// base first (§3.14.2); then children, one-shot init, mode transition, stall watch
METHOD PROTECTED OnCyclic : DINT
VAR
    publishIdx : INT;
    modeIdx    : E_Mode;
    styleIdx   : E_RunStyle;
    previousMode : E_Mode;
    modeExitResult : DINT;
END_VAR
OnCyclic := SUPER^.OnCyclic();
_M_TickChildren();
_M_OeeUpdate();                                       // §8.5.1 time accounting + sampling
AlarmLog.Cyclic();                                    // §8.10 shelf auto-expiry
_M_HandleHmiRequest();                                // §3.10 request mailbox
Access.Cyclic();
// §9.8 data-driven Control On/Off request endpoint. Off wins if both arrive;
// the domain/power-group implementation still validates safety, health and rearm.
ControlOnRequest := FALSE;
ControlOffRequest := FALSE;
IF ReqControlOff THEN
    ReqControlOff := FALSE;
    ReqControlOn := FALSE;
    IF Access.PermitsLogged(Gate := E_GatedAction.POWER_CONTROL) THEN
        ControlOffRequest := TRUE;
    END_IF
ELSIF ReqControlOn THEN
    ReqControlOn := FALSE;
    IF Access.PermitsLogged(Gate := E_GatedAction.POWER_CONTROL) THEN
        ControlOnRequest := TRUE;
    END_IF
END_IF
// §3.14.4 — pending mode change; §3.4.1 style decides graceful vs immediate
IF _modePend THEN
    IF _exec = E_ExecState.BUSY THEN
        IF ModePolicy[TO_INT(_mode)].Style = E_ModeSwitchStyle.GRACEFUL THEN
            _stopReq := TRUE;                             // finish the cycle at its stop point
        ELSE
            modeExitResult := OnModeExit(FirstCall := _modeExitFirst,
                RequestedMode := _modeReq);
            _modeExitFirst := FALSE;
            IF modeExitResult = 0 THEN
                OnAbort();                                // IMMEDIATE: cancel now (override may defer)
            END_IF
        END_IF
    ELSE
        IF _exec <> E_ExecState.READY THEN
            Execute := FALSE;                             // release the run command (§6.1 reset)
        ELSE
            previousMode := _mode;
            _mode := _modeReq;
            _modePend := FALSE;
            _modeExitFirst := FALSE;
            _M_CascadeMode(_mode);                        // §3.7 cascade [TC3]
            OnModeChanged(NewMode := _mode, OldMode := previousMode);
        END_IF
    END_IF
END_IF
// §8.3(c) — automatic fault capture: ERROR entry raises, ERROR exit marks gone
IF (_exec = E_ExecState.ERROR) AND (_faultEvt = 0) THEN
    _faultEvt := AlarmLog.RaiseDiag(D := _diag, ResetClass := E_ResetClass.MANUAL_RESET);
    _M_PartAborted();                  // §3.16.3: a faulted part leaves without a valid result
ELSIF (_exec <> E_ExecState.ERROR) AND (_faultEvt > 0) THEN
    AlarmLog.Gone(Slot := _faultEvt);                            // -> WAIT_RESET (blocking)
    _faultEvt := 0;
END_IF
// §6.9 — instant rollup on awaited Error; stall as PENDING otherwise
IF _exec = E_ExecState.BUSY THEN
    IF (_awaits <> 0) AND_THEN _awaits.FaultActive THEN
        _M_FaultDiag(_awaits.GetFaultSummary());
    ELSE
        _tStall(IN := TRUE, PT := SEL(CurrentStep.ExpectedTime > T#0S, StallTime, CurrentStep.ExpectedTime));
        IF _tStall.Q THEN
            _M_StallWalk();
        END_IF
    END_IF
ELSE
    _tStall(IN := FALSE);
END_IF
// §6.9(a) — every new fault joins the shift-change ring, no historian needed
_fTrig(CLK := (_exec = E_ExecState.ERROR));
IF _fTrig.Q THEN
    _M_PushHistory(_diag);
END_IF
// §8.11.4(d) — creeping WORK time is a MAINTENANCE event (Low), not downtime:
// the profiler pulses once per excursion past the configured baseline band.
IF Profiler.DegradedTrig THEN
    _M_RaiseMaintenance(Reason := E_Reason.CYCLE_TIME_DEGRADED,
        Text := 'std.maintenance.cycleTimeDegraded');
END_IF
ModeActivePublished := _mode;
RunningPublished := (_exec = E_ExecState.BUSY);
StopPendingPublished := _stopReq AND (_exec = E_ExecState.BUSY);
FOR publishIdx := 0 TO PL_Fraktal.MODE_COUNT - 1 DO
    modeIdx := publishIdx;
    SupportedModesPublished[publishIdx] := _M_Supports(Mode := modeIdx);
END_FOR
FOR publishIdx := 0 TO 2 DO
    styleIdx := publishIdx;
    SupportedRunStylesPublished[publishIdx] := _M_SupportsRunStyle(Style := styleIdx);
END_FOR
END_METHOD

// §3.14 hook — one-shot after first operational scan
METHOD PROTECTED OnInit : DINT
OnInit := SUPER^.OnInit();
Access.Setup(Provider := 0, pAlarmLog := ADR(AlarmLog)); // preserves an injected provider
_M_InitModePolicy();
// §3.10.2 — seed the manifest revision from boot time so every PLC restart or
// re-activation yields a NEW value (a plain counter would repeat after reboot
// and an HMI could keep a stale manifest undetected). Config writes increment.
ConfigRev := DT_TO_UDINT(F_Now());
END_METHOD

// §3.14 hook — after the new mode is committed
METHOD PROTECTED OnModeChanged : DINT
VAR_INPUT
    NewMode : E_Mode;
    OldMode : E_Mode;
END_VAR
OnModeChanged := 0;
END_METHOD

// §3.14.4 — called every scan while a mode request is pending and the Unit is BUSY.
// Return 0 = consent to immediate cancel (default); >0 = still stopping gracefully.
METHOD PROTECTED OnModeExit : DINT
VAR_INPUT
    FirstCall : BOOL;
    RequestedMode : E_Mode;
END_VAR
OnModeExit := 0;
END_METHOD

// §8.3(b) — deliberate operator reset of blocking events (release-gated per §7.6/§14).
// Closes WAIT_RESET events; an event whose condition persists stays ACTIVE.
METHOD OperatorReset : BOOL
IF NOT Access.PermitsLogged(Gate := E_GatedAction.ALARM_RESET) THEN
    OperatorReset := FALSE;            // §7.7
    RETURN;
END_IF
OperatorReset := AlarmLog.OperatorReset();
END_METHOD

// §3.8 optional HMI/MES selection catalog. Recipe providers remain pluggable;
// the application registers only the model identities it deliberately exposes.
METHOD RegisterAvailableModel : BOOL
VAR_INPUT
    Id : ST_ModelId;
END_VAR
VAR
    i : INT;
END_VAR
RegisterAvailableModel := FALSE;
IF (Id.ModelCode = '') OR (AvailableModelCount >= PL_Fraktal.MAX_RECIPES) THEN
    RETURN;
END_IF
FOR i := 1 TO AvailableModelCount DO
    IF AvailableModels[i].ModelCode = Id.ModelCode THEN
        RETURN;
    END_IF
END_FOR
AvailableModelCount := AvailableModelCount + 1;
AvailableModels[AvailableModelCount] := Id;
ConfigRev := ConfigRev + 1;    // §3.10.2 — manifest changed
RegisterAvailableModel := TRUE;
END_METHOD

// Core §7.8 — full rollup for the simpler gated Unit actions (Stop, ALARM_RESET,
// CHANGEOVER, MODE_CHANGE, step). Same predicate the gates use. Start has its own
// richer ReleaseReportStart (interlocks); manual has ReleaseReportManual (target).
METHOD ReleaseReportAction : BOOL
VAR_INPUT
    Gate : E_GatedAction;
END_VAR
VAR_IN_OUT
    Report : ST_ReleaseReport;
END_VAR
Report.Count := 0;
Report.Released := FALSE;
// access is the common gate
IF NOT Access.Permits(Gate := Gate) THEN
    _M_AddReason(Report := Report, Text := 'std.release.insufficientAction', Reason := E_Reason.NONE, Kind := E_ReleaseKind.ACCESS);
END_IF
// per-action state preconditions
CASE Gate OF
    E_GatedAction.CHANGEOVER:
        IF _exec = E_ExecState.BUSY THEN
            _M_AddReason(Report := Report, Text := 'std.release.changeoverRunning', Reason := E_Reason.NONE, Kind := E_ReleaseKind.MODE);
        END_IF
    E_GatedAction.ALARM_RESET:
        IF NOT AlarmLog.Blocking THEN
            _M_AddReason(Report := Report, Text := 'std.release.noBlockingAlarm', Reason := E_Reason.NONE, Kind := E_ReleaseKind.OTHER);
        END_IF
    E_GatedAction.MODE_CHANGE:
        IF _modePend THEN
            _M_AddReason(Report := Report, Text := 'std.release.modeChangeAlreadyPending', Reason := E_Reason.NONE, Kind := E_ReleaseKind.MODE);
        END_IF
ELSE
    ;                                          // actions with no extra state predicate
END_CASE
Report.Released := (Report.Count = 0);
ReleaseReportAction := Report.Released;
END_METHOD

// Core §7.8 — full rollup of why a manual command to Target would be refused (§7.6.1).
METHOD ReleaseReportManual : BOOL
VAR_INPUT
    TargetPath : STRING(255);
    Value : DINT;
END_VAR
VAR_IN_OUT
    Report : ST_ReleaseReport;
END_VAR
Report.Count := 0;
Report.Released := FALSE;
IF _mode <> E_Mode.MANUAL THEN
    _M_AddReason(Report := Report, Text := 'std.release.manualModeRequired', Reason := E_Reason.NONE, Kind := E_ReleaseKind.MODE);
END_IF
IF NOT Access.Permits(Gate := E_GatedAction.MANUAL) THEN
    _M_AddReason(Report := Report, Text := 'std.release.insufficientManual', Reason := E_Reason.NONE, Kind := E_ReleaseKind.ACCESS);
END_IF
_M_AppendManualInterlocks(TargetPath := TargetPath, Value := Value, Report := Report);  // §7.6, target+command-aware
Report.Released := (Report.Count = 0);
ReleaseReportManual := Report.Released;
END_METHOD

// Core §7.8 — pure query: the FULL rollup of why Start would be refused right now.
// This is the authoritative machine predicate consumed by Start (no drift).
// Released = TRUE means Start proceeds. Lists mode + access + blocking-alarm,
// control-domain, and concrete mode-entry release reasons. The caller owns the
// bounded report storage; returning this large record by value can overflow a
// TwinCAT task stack when Start consumes the result.
METHOD ReleaseReportStart : BOOL
VAR_IN_OUT
    Report : ST_ReleaseReport;
END_VAR
Report.Count := 0;
Report.Released := FALSE;
// access (§7.7)
IF NOT Access.Permits(Gate := E_GatedAction.START_STOP) THEN
    _M_AddReason(Report := Report, Text := 'std.release.insufficientStartStop', Reason := E_Reason.NONE, Kind := E_ReleaseKind.ACCESS);
END_IF
// mode / run state (§3.4)
IF _modePend THEN
    _M_AddReason(Report := Report, Text := 'std.release.modeChangePending', Reason := E_Reason.NONE, Kind := E_ReleaseKind.MODE);
END_IF
IF _mode = E_Mode.MANUAL THEN
    _M_AddReason(Report := Report, Text := 'std.release.manualHasNoAutoSequence', Reason := E_Reason.NONE, Kind := E_ReleaseKind.MODE);
END_IF
IF _exec <> E_ExecState.READY THEN
    _M_AddReason(Report := Report, Text := 'std.release.unitNotReady', Reason := E_Reason.NONE, Kind := E_ReleaseKind.MODE);
END_IF
// blocking alarm (§8.3)
IF AlarmLog.Blocking THEN
    _M_AddReason(Report := Report, Text := 'std.release.manualReset', Reason := E_Reason.NONE, Kind := E_ReleaseKind.ALARM);
END_IF
IF ControlDomain.Present AND NOT ControlDomain.ReadyForStart THEN
    _M_AddReason(Report := Report, Text := 'std.release.controlDomainNotReady', Reason := E_Reason.NONE, Kind := E_ReleaseKind.INTERLOCK);
END_IF
// active mode's immediate entry/frontier conditions (concrete override)
_M_AppendInterlocks(Report := Report);
Report.Released := (Report.Count = 0);
ReleaseReportStart := Report.Released;
END_METHOD

// §8.5.1 — clear accumulators + ring (shift start). Gated: §7.7 DATA_WRITE; audited §8.3.
METHOD ResetOee : BOOL
VAR
    i : INT;
    auditSlot : INT;
END_VAR
IF NOT Access.PermitsLogged(Gate := E_GatedAction.DATA_WRITE) THEN
    ResetOee := FALSE;
    RETURN;
END_IF
Oee.RunMs := 0; Oee.DownMs := 0; Oee.IdleMs := 0;
FOR i := 1 TO PL_Fraktal.MAX_OEE_SAMPLES DO
    OeeTrend[i].Oee := 0.0; OeeTrend[i].OeeValid := FALSE;
    OeeTrend[i].Availability := 0.0; OeeTrend[i].Performance := 0.0; OeeTrend[i].Quality := 0.0;
END_FOR
OeeTrendHead := 0;
_oeeSampMs := 0;
_M_OeeCompute();
auditSlot := AlarmLog.Raise(Reason := E_Reason.NONE,
    Text := 'std.audit.oeeReset', Source := _name,
    Severity := E_Severity.LOW, Category := E_Category.SYSTEM, ResetClass := E_ResetClass.AUTO_RESET);
IF auditSlot > 0 THEN AlarmLog.Gone(Slot := auditSlot); END_IF
ResetOee := TRUE;
END_METHOD

// §3.4.2 — HMI HOLD_TO_RUN input. NON-SAFETY (§9): never a dead-man; interlocks
// still apply at every step. TRUE only while the operator holds the button.
METHOD SetHoldRun : BOOL
VAR_INPUT
    Held : BOOL;
END_VAR
IF Held AND (NOT Access.PermitsLogged(Gate := E_GatedAction.START_STOP)
OR (RunStyle <> E_RunStyle.HOLD_TO_RUN) OR (_exec <> E_ExecState.BUSY)) THEN
    SetHoldRun := FALSE;
    RETURN;
END_IF
_holdRun := Held;                     // FALSE is always accepted so a hold cannot stick
SetHoldRun := TRUE;
END_METHOD

// §8.5.1 — configure the ideal cycle time (per model, §3.8). 0 disables Performance.
METHOD SetIdealCycle : BOOL
VAR_INPUT
    Ms : UDINT;
END_VAR
Oee.IdealCycleMs := Ms;
SetIdealCycle := TRUE;
END_METHOD

// §3.4/§3.7 — FALSE = unsupported (graceful rejection); TRUE = committed or pending
METHOD SetMode : BOOL
VAR_INPUT
    Mode : E_Mode;
END_VAR
IF NOT Access.PermitsLogged(Gate := E_GatedAction.MODE_CHANGE) THEN
    SetMode := FALSE;                  // §7.7(c): who-gate ANDs the machine gates
    RETURN;
END_IF
IF NOT _M_Supports(Mode) THEN
    SetMode := FALSE;
    RETURN;
END_IF
IF (Mode = _mode) AND NOT _modePend THEN
    SetMode := TRUE;
    RETURN;
END_IF
// §3.4.1 shield: policy of the mode being LEFT governs while its sequence runs
IF (_exec = E_ExecState.BUSY)
AND (ModePolicy[TO_INT(_mode)].Shield = E_ModeSwitchShield.BLOCKED_WHILE_RUNNING) THEN
    SetMode := FALSE;                  // must Stop first (graceful rejection, not a fault)
    RETURN;
END_IF
IF (NOT _modePend) OR (_modeReq <> Mode) THEN
    _modeExitFirst := TRUE;
END_IF
_modeReq := Mode;
_modePend := TRUE;
SetMode := TRUE;
END_METHOD

// §3.1b/§3.8 — transactional model change: prepare the whole subtree, then commit.
METHOD SetModel : BOOL
VAR_INPUT
    Id : ST_ModelId;
END_VAR
IF NOT Access.PermitsLogged(Gate := E_GatedAction.CHANGEOVER) THEN
    SetModel := FALSE;                 // §7.7
    RETURN;
END_IF
IF _exec = E_ExecState.BUSY THEN
    SetModel := FALSE;                 // changeover is not mid-cycle (§3.8 loads at CHANGEOVER)
    RETURN;
END_IF
IF NOT PrepareRecipe(Model := Id) THEN
    AbortRecipe();
    SetModel := FALSE;
    RETURN;
END_IF
CommitRecipe();                         // infallible after successful preparation
Model := Id;                           // identity changes only after subtree commit
ConfigRev := ConfigRev + 1;            // §3.10.2 — recipe/config leaves changed
SetModel := TRUE;
END_METHOD

// §3.16.2 — inject the part carrier at the composition root (0 = traceability off).
// Source-agnostic: BY_POSITION local, RFID, DataMatrix, or host, behind I_PartCarrier.
METHOD SetPartCarrier : BOOL
VAR_INPUT
    Carrier : I_PartCarrier;
END_VAR
_carrier := Carrier;
SetPartCarrier := (Carrier <> 0);
END_METHOD

// §3.4.2 — HMI selects the run style for the active mode. Modes that don't opt in
// (see _M_SupportsRunStyle) reject non-CONTINUOUS. Access: MODE_CHANGE-gated (§7.7).
METHOD SetRunStyle : BOOL
VAR_INPUT
    Style : E_RunStyle;
END_VAR
IF NOT Access.PermitsLogged(Gate := E_GatedAction.MODE_CHANGE) THEN
    SetRunStyle := FALSE;
    RETURN;
END_IF
IF (Style <> E_RunStyle.CONTINUOUS) AND NOT _M_SupportsRunStyle(Style := Style) THEN
    SetRunStyle := FALSE;               // mode didn't opt into stepping (graceful reject)
    RETURN;
END_IF
RunStyle := Style;
SetRunStyle := TRUE;
END_METHOD

// §8.10 — gated HMI entry: shelve an active alarm's ANNUNCIATION (control untouched).
// §7.7 ALARM_SHELVE + audit; refuses SAFETY / unrationalized reasons (AlarmLog rules).
METHOD ShelveAlarm : BOOL
VAR_INPUT
    Slot      : INT;
    DurationS : UDINT;
END_VAR
IF NOT Access.PermitsLogged(Gate := E_GatedAction.ALARM_SHELVE) THEN
    ShelveAlarm := FALSE;
    RETURN;
END_IF
ShelveAlarm := AlarmLog.Shelve(Slot := Slot, DurationS := DurationS);
END_METHOD

// §3.3/§6 intro — the run IS a §6.1 command.
// §7.8: ReleaseReportStart is the authoritative machine gate as well as the
// operator explanation, so a concrete Unit cannot report an interlock it ignores.
// Build directly into the published response storage: ST_ReleaseReport is too
// large for nested by-value/local copies on a small TwinCAT task stack.
METHOD Start : BOOL
IF NOT Access.PermitsLogged(Gate := E_GatedAction.START_STOP) THEN
    Start := FALSE;                    // §7.7
    RETURN;
END_IF
IF ReleaseReportStart(Report := HmiResponse.Report) THEN
    _stopReq := FALSE;                 // §8.3(b): a MANUAL_RESET event blocks restart
    Execute := TRUE;
    Start := TRUE;
ELSE
    Start := FALSE;
END_IF
END_METHOD

// §3.4.2 — HMI single-step: request advance of one step (edge-consumed by _M_StepGate).
METHOD StepRequest : BOOL
IF NOT Access.PermitsLogged(Gate := E_GatedAction.START_STOP)
OR (RunStyle <> E_RunStyle.SINGLE_STEP) OR (_exec <> E_ExecState.BUSY) THEN
    StepRequest := FALSE;
    RETURN;
END_IF
_stepReq := TRUE;
StepRequest := TRUE;
END_METHOD

// §3.3 — stop after the current cycle
METHOD Stop : BOOL
IF NOT Access.PermitsLogged(Gate := E_GatedAction.START_STOP) THEN
    Stop := FALSE;                     // §7.7
    RETURN;
END_IF
IF _exec = E_ExecState.BUSY THEN
    _stopReq := TRUE;
ELSE
    _stopReq := FALSE;
    Execute := FALSE;                  // release a terminal run command (ERROR/DONE/ABORTED)
END_IF
Stop := TRUE;
END_METHOD

// §3.4 — TRUE while a stop is requested but the sequence is still finishing
// (running -> stopping). HMI blinks the stop button on this.
PROPERTY StopPending : BOOL
GET
StopPending := _stopReq AND (_exec = E_ExecState.BUSY);
END_GET
END_PROPERTY

// §8.10 — gated HMI entry: restore annunciation.
METHOD UnshelveAlarm : BOOL
VAR_INPUT
    Slot : INT;
END_VAR
IF NOT Access.PermitsLogged(Gate := E_GatedAction.ALARM_SHELVE) THEN
    UnshelveAlarm := FALSE;
    RETURN;
END_IF
UnshelveAlarm := AlarmLog.Unshelve(Slot := Slot);
END_METHOD

END_FUNCTION_BLOCK

// ---- Connectivity/F_AppendTopologyConfig.TcPOU
// Core §3.10.2/§10.5.1 — export the activation-static fieldbus identity (tags,
// addresses, wiring, hierarchy) into the config manifest. The live members
// (State/LinkOk/values/force/quality/fault) stay cyclically published; the
// static members carry OPC.UA.DA=0 in ST_BusNode/ST_IoChannel and reach the
// HMI only through this walk. Item fragments use the server's array naming
// (Nodes/Nodes[i]/..., Channels/Channels[j]/...) under the reserved scope
// '#Fieldbus' so a generic client can rebuild the exact browse paths.
// Only populated slots are exported — the empty tail of the bounded table
// costs nothing on the wire.
FUNCTION F_AppendTopologyConfig : BOOL
VAR_IN_OUT
    Topology : ST_FieldbusTopology;
    Pager    : FB_ConfigPager;
END_VAR
VAR
    i, j       : INT;
    nodeBase   : STRING(255);
    chanBase   : STRING(255);
    item       : STRING(255);
END_VAR
VAR CONSTANT
    SCOPE_FIELDBUS : STRING(16) := '#Fieldbus';
END_VAR

F_AppendTopologyConfig := TRUE;
FOR i := 1 TO Topology.NodeCount DO
    IF (i < 1) OR (i > PL_Fraktal.MAX_BUS_NODES) THEN
        EXIT;                                       // defensive bound (§5.6)
    END_IF
    nodeBase := CONCAT('Nodes/Nodes[', CONCAT(TO_STRING(i), ']/'));
    Pager.M_Append(Scope := SCOPE_FIELDBUS,
        Item := CONCAT(nodeBase, 'Name'), ValueText := Topology.Nodes[i].Name);
    Pager.M_Append(Scope := SCOPE_FIELDBUS,
        Item := CONCAT(nodeBase, 'DescriptionKey'),
        ValueText := Topology.Nodes[i].DescriptionKey);
    Pager.M_Append(Scope := SCOPE_FIELDBUS,
        Item := CONCAT(nodeBase, 'TypeId'), ValueText := Topology.Nodes[i].TypeId);
    Pager.M_Append(Scope := SCOPE_FIELDBUS,
        Item := CONCAT(nodeBase, 'Address'), ValueText := Topology.Nodes[i].Address);
    Pager.M_AppendNumber(Scope := SCOPE_FIELDBUS,
        Item := CONCAT(nodeBase, 'ParentIdx'),
        Number := TO_DINT(Topology.Nodes[i].ParentIdx));
    Pager.M_AppendNumber(Scope := SCOPE_FIELDBUS,
        Item := CONCAT(nodeBase, 'ChannelCount'),
        Number := TO_DINT(Topology.Nodes[i].ChannelCount));
    FOR j := 1 TO Topology.Nodes[i].ChannelCount DO
        IF (j < 1) OR (j > PL_Fraktal.MAX_NODE_CHANNELS) THEN
            EXIT;                                   // defensive bound (§5.6)
        END_IF
        chanBase := CONCAT(nodeBase,
            CONCAT('Channels/Channels[', CONCAT(TO_STRING(j), ']/')));
        Pager.M_Append(Scope := SCOPE_FIELDBUS,
            Item := CONCAT(chanBase, 'Name'),
            ValueText := Topology.Nodes[i].Channels[j].Name);
        Pager.M_Append(Scope := SCOPE_FIELDBUS,
            Item := CONCAT(chanBase, 'DescriptionKey'),
            ValueText := Topology.Nodes[i].Channels[j].DescriptionKey);
        Pager.M_Append(Scope := SCOPE_FIELDBUS,
            Item := CONCAT(chanBase, 'Address'),
            ValueText := Topology.Nodes[i].Channels[j].Address);
        Pager.M_Append(Scope := SCOPE_FIELDBUS,
            Item := CONCAT(chanBase, 'Path'),
            ValueText := Topology.Nodes[i].Channels[j].Path);
        Pager.M_Append(Scope := SCOPE_FIELDBUS,
            Item := CONCAT(chanBase, 'ModulePath'),
            ValueText := Topology.Nodes[i].Channels[j].ModulePath);
        Pager.M_AppendNumber(Scope := SCOPE_FIELDBUS,
            Item := CONCAT(chanBase, 'Dir'),
            Number := TO_DINT(Topology.Nodes[i].Channels[j].Dir));
        Pager.M_AppendNumber(Scope := SCOPE_FIELDBUS,
            Item := CONCAT(chanBase, 'Kind'),
            Number := TO_DINT(Topology.Nodes[i].Channels[j].Kind));
        Pager.M_Append(Scope := SCOPE_FIELDBUS,
            Item := CONCAT(chanBase, 'Unit'),
            ValueText := Topology.Nodes[i].Channels[j].Unit);
    END_FOR
END_FOR

END_FUNCTION

// ---- Connectivity/FB_DeviceConnectorBase.TcPOU
// Core §3.15 written once: session + heartbeat + LinkTimeout loss confirm +
// bounded exponential backoff reconnect + NO self-resume of dependents (that is
// the fronting CM's contract). A transport implements only _M_Open/_M_Close/
// _M_HbStart/_M_HbPoll. Row T7 of §5.7 is proven here once.
FUNCTION_BLOCK ABSTRACT FB_DeviceConnectorBase IMPLEMENTS I_DeviceConnector
VAR_INPUT
    HbPeriod    : TIME := T#1S;
    LinkTimeout : TIME := T#3S;
    BackoffMin  : TIME := T#500MS;
    BackoffMax  : TIME := T#10S;
    Reaction    : E_LinkReaction := E_LinkReaction.HOLD;   // consumed by the fronting CM
END_VAR
VAR
    _name      : STRING(80);
    _sessionUp : BOOL;
    _linked    : BOOL;
    _hbBusy    : BOOL;
    _lastSeen  : DT;
    _diag      : ST_Diagnostic;
    _tHb, _tLoss, _tBk : TON;
    _backoffMs : DINT;
END_VAR

Cyclic();

METHOD Connect : BOOL
Connect := _M_TryOpen();
END_METHOD

METHOD Cyclic : BOOL
IF NOT _sessionUp THEN
    // bounded exponential backoff (§3.15) — never a tight reconnect loop
    _tBk(IN := TRUE, PT := DINT_TO_TIME(_backoffMs));
    IF _tBk.Q THEN
        _tBk(IN := FALSE);
        IF NOT _M_TryOpen() THEN
            _backoffMs := MIN(_backoffMs * 2, TIME_TO_DINT(BackoffMax));
        END_IF
    END_IF
    Cyclic := TRUE;
    RETURN;
END_IF
// heartbeat: issue when due, poll while busy
IF NOT _hbBusy THEN
    _tHb(IN := TRUE, PT := HbPeriod);
    IF _tHb.Q THEN
        _tHb(IN := FALSE);
        _hbBusy := _M_HbStart();
    END_IF
ELSE
    CASE _M_HbPoll() OF
        E_HbResult.OK:
            _hbBusy := FALSE;
            _linked := TRUE;
            _lastSeen := F_Now();                 // §2.7
            _diag.ReasonCode := E_Reason.NONE;
            _diag.Description := '';
            _tLoss(IN := FALSE);                  // healthy beat resets loss confirm
        E_HbResult.FAIL:
            _hbBusy := FALSE;
            _M_Lost(E_Reason.DEVICE_PROTOCOL_ERROR, 'std.error.heartbeatBadReply');
            Cyclic := TRUE;
            RETURN;
        E_HbResult.PENDING:
            ;                                      // request still in flight
    ELSE
        _hbBusy := FALSE;
        _M_Lost(E_Reason.DEVICE_PROTOCOL_ERROR, 'std.error.heartbeatResultInvalid');
        Cyclic := TRUE;
        RETURN;
    END_CASE
END_IF
// confirm loss only after LinkTimeout without a healthy beat (§3.15.2)
_tLoss(IN := TRUE, PT := LinkTimeout);
IF _tLoss.Q THEN
    _M_Lost(E_Reason.LINK_TIMEOUT, 'std.error.heartbeatLapsed');
END_IF
Cyclic := TRUE;
END_METHOD

METHOD Disconnect : BOOL
_M_Close();
_sessionUp := FALSE;
_linked := FALSE;
Disconnect := TRUE;
END_METHOD

METHOD GetFaultSummary : ST_Diagnostic
GetFaultSummary := _diag;
END_METHOD

METHOD PrepareRecipe : BOOL
VAR_INPUT
    Model : ST_ModelId;
END_VAR
PrepareRecipe := TRUE;
END_METHOD

METHOD CommitRecipe
END_METHOD

METHOD AbortRecipe
END_METHOD

METHOD Setup : BOOL
VAR_INPUT
    Name : STRING(80);
END_VAR
_name := Name;
_backoffMs := TIME_TO_DINT(BackoffMin);
Setup := TRUE;
END_METHOD

METHOD PROTECTED ABSTRACT _M_Close : BOOL
END_METHOD

// PENDING while in flight; OK resets loss confirm; FAIL = protocol error
METHOD PROTECTED ABSTRACT _M_HbPoll : E_HbResult
END_METHOD

METHOD PROTECTED ABSTRACT _M_HbStart : BOOL
END_METHOD

// stamp the link first-out, drop the session; reconnection is backoff-bounded,
// resumption of dependent commands is NEVER automatic (§3.15/§9.3)
METHOD PROTECTED _M_Lost
VAR_INPUT
    Reason : E_Reason;
    Text   : STRING(255);
END_VAR
IF _diag.ReasonCode <> Reason THEN
    _diag.Since := F_Now();
END_IF
_diag.ReasonCode  := Reason;
_diag.Description := Text;
_diag.SourcePath  := _name;
_diag.Severity    := E_Severity.MED;
_diag.Category    := E_Category.SYSTEM;
_linked := FALSE;
_hbBusy := FALSE;
_M_Close();
_sessionUp := FALSE;
END_METHOD

METHOD PROTECTED ABSTRACT _M_Open : BOOL
END_METHOD

METHOD PROTECTED _M_TryOpen : BOOL
IF _M_Open() THEN
    _sessionUp := TRUE;
    _backoffMs := TIME_TO_DINT(BackoffMin);
    _M_TryOpen := TRUE;
ELSE
    _M_TryOpen := FALSE;
END_IF
END_METHOD

PROPERTY FaultActive : BOOL
GET
FaultActive := (NOT _linked) AND (_diag.ReasonCode <> E_Reason.NONE);
END_GET
END_PROPERTY

PROPERTY LastSeen : DT
GET
LastSeen := _lastSeen;
END_GET
END_PROPERTY

PROPERTY Linked : BOOL
GET
Linked := _linked;
END_GET
END_PROPERTY

PROPERTY LinkReason : ST_Diagnostic
GET
LinkReason := _diag;
END_GET
END_PROPERTY

PROPERTY ModuleType : E_ModuleType
GET
ModuleType := E_ModuleType.CONTROL_MODULE;
END_GET
END_PROPERTY

PROPERTY Name : STRING(80)
GET
Name := _name;
END_GET
END_PROPERTY

PROPERTY State : E_ExecState
GET
State := SEL(FaultActive, E_ExecState.READY, E_ExecState.ERROR);
END_GET
END_PROPERTY

END_FUNCTION_BLOCK

// ---- Connectivity/FB_EcBusHealth.TcPOU
// Core §10.5.1 infrastructure service: read the REAL, live state of every
// EtherCAT slave directly from the fieldbus master (Tc2_EtherCAT) and publish it
// per node, so the HMI fieldbus tree mirrors XAE — independent of any Control-On
// or safety verdict. Auto-detects from hardware: the project supplies only the
// master AmsNetId ('' = local CPU) and how its topology node indices line up
// with the master's slave ordering (one offset), not per-node wiring.
//
// This is not a module tier and owns no process image. It calls
// FB_IoTopologyPublisher.M_SetNodeState for each mapped node.
FUNCTION_BLOCK FB_EcBusHealth
VAR
    {attribute 'OPC.UA.DA' := '0'}
    _pub : POINTER TO FB_IoTopologyPublisher;
    _netId : T_AmsNetId;          // EtherCAT MASTER device AmsNetId (see Setup)
    _firstSlaveNode : INT;        // topology node index of master slave #1
    _slaveCount : INT;            // topology nodes that are real EtherCAT slaves
    _masterNode : INT;            // topology node index of the master itself (0 = none)
    _attached : BOOL;

    // Auto-detection of the EtherCAT master's AmsNetId (no project wiring): the
    // master's NetId is the local AMS NetId with the last two bytes replaced by
    // 2.1 (Beckhoff convention -- a PC 'a.b.c.d.1.1' has its EtherCAT master at
    // 'a.b.c.d.2.1'; the InfoSys FB_EcGetAllSlaveStates example uses exactly this
    // pairing). Overridable via Setup for non-standard configurations.
    {attribute 'OPC.UA.DA' := '0'}
    _fbLocalNetId : Tc2_Utilities.FB_GetLocalAmsNetId;
    _autoDetect : BOOL;           // TRUE = derive the master NetId at runtime
    {attribute 'OPC.UA.DA' := '0'}
    _netIdArr : T_AmsNetIdArr;    // scratch for the derived master NetId

    {attribute 'OPC.UA.DA' := '0'}
    _fbStates : Tc2_EtherCAT.FB_EcGetAllSlaveStates;
    // Bounded state buffer, one ST_EcSlaveState (deviceState + linkState) per
    // slave. Beckhoff declares pStateBuf as ARRAY[0..EC_MAX_SLAVES], so this
    // buffer is ZERO-BASED: slave i (1..n, master scan order) is _stateBuf[i-1].
    {attribute 'OPC.UA.DA' := '0'}
    _stateBuf : ARRAY[0..PL_Fraktal.MAX_BUS_NODES] OF Tc2_EtherCAT.ST_EcSlaveState;
    _step : INT;
    _tPoll : TON;
END_VAR
VAR_OUTPUT
    // Diagnostics so a fieldbus read failure is visible instead of silently
    // showing every node as faulted. Published for the HMI/engineer.
    ReadOk : BOOL;                // last slave-state read succeeded
    LastErrorId : UDINT;          // ADS error of the last failed read (0 = none)
    SlavesReported : UINT;        // slaves the master reports (nSlaves output)
    NetIdMissing : BOOL;          // TRUE = InfoData.AmsNetId not linked (all zero)
    MasterNetId : T_AmsNetId;     // the resolved master NetId actually being used
END_VAR

;

// Bind the publisher and describe how topology nodes map to master slaves.
// MasterNetIdArr = OPTIONAL override for the EtherCAT master's AmsNetId. Pass all
//   zeros (the normal case, e.g. an unassigned T_AmsNetIdArr) to AUTO-DETECT it at
//   runtime: the library reads the local AMS NetId and applies the Beckhoff master
//   convention (last two bytes -> 2.1), so no project wiring, no XAE checkbox and
//   no hand-typed address are needed. Supply a value only for a non-standard
//   configuration (e.g. a remote master, or several masters on one PC), typically
//   by linking that master's InfoData.AmsNetId.
// FirstSlaveNode = topology index of the first EtherCAT slave (the coupler);
// SlaveCount = number of consecutive topology nodes that are real slaves, in
// master scan order; MasterNodeIndex = topology index of the EtherCAT master
// itself, or 0 if not represented.
METHOD Setup : BOOL
VAR_INPUT
    Publisher : REFERENCE TO FB_IoTopologyPublisher;
    MasterNetIdArr : T_AmsNetIdArr;
    FirstSlaveNode : INT;
    SlaveCount : INT;
    MasterNodeIndex : INT;
END_VAR
VAR
    i : INT;
    anyNonZero : BOOL;
END_VAR
// All-zero (or omitted) = auto-detect; any explicit value is used verbatim.
anyNonZero := FALSE;
FOR i := 0 TO 5 DO
    IF MasterNetIdArr[i] <> 0 THEN
        anyNonZero := TRUE;
    END_IF
END_FOR

_attached := __ISVALIDREF(Publisher)
    AND (FirstSlaveNode >= 1)
    AND (SlaveCount >= 0)
    AND (SlaveCount <= PL_Fraktal.MAX_BUS_NODES);
IF _attached THEN
    _pub := ADR(Publisher);
    _autoDetect := NOT anyNonZero;
    IF anyNonZero THEN
        // Tc2_System helper: byte array -> 'a.b.c.d.e.f' string.
        _netId := Tc2_System.F_CreateAmsNetId(nIds := MasterNetIdArr);
        MasterNetId := _netId;
        NetIdMissing := FALSE;
        _step := 0;
    ELSE
        // Resolve the local NetId first (step -10), then start polling.
        _netId := '';
        MasterNetId := '';
        NetIdMissing := TRUE;   // cleared once auto-detection succeeds
        _step := -10;
    END_IF
    _firstSlaveNode := FirstSlaveNode;
    _slaveCount := SlaveCount;
    _masterNode := MasterNodeIndex;
END_IF
Setup := _attached;
END_METHOD

// Non-blocking cyclic refresh: (re)issue the slave-state read at a bounded rate,
// then publish each node's real state. On a read error every mapped node is
// marked OFFLINE (fail-visible: an unreachable master is not "operational").
METHOD M_Refresh
VAR
    i : INT;
    node : INT;
    mapped : E_NodeState;
    linkOk : BOOL;
END_VAR
IF NOT _attached THEN
    RETURN;
END_IF

// Drive the async read. Re-trigger on a slow poll so a stuck call cannot pin the
// task; FB_EcGetAllSlaveStates is edge-triggered by bExecute. The slave count is
// implied by cbBufLen (nSlave * SIZEOF(ST_EcSlaveState)); there is no count input.
CASE _step OF
    -10:
        // Auto-detect: ask the router for this PC's AmsNetId.
        _fbLocalNetId(bExecute := FALSE);
        _fbLocalNetId(bExecute := TRUE);
        _step := -5;
    -5:
        _fbLocalNetId(bExecute := FALSE);
        IF NOT _fbLocalNetId.bBusy THEN
            IF _fbLocalNetId.bError THEN
                // Cannot resolve: stay fail-visible and retry on the next poll.
                ReadOk := FALSE;
                LastErrorId := _fbLocalNetId.nErrId;
                NetIdMissing := TRUE;
                _M_PublishAllOffline();
                _step := -10;
            ELSE
                // Beckhoff convention: the EtherCAT master of a PC 'a.b.c.d.1.1'
                // is 'a.b.c.d.2.1'. Keep the first four bytes, force 2.1.
                _netIdArr := _fbLocalNetId.AddrBytes;
                _netIdArr[4] := 2;
                _netIdArr[5] := 1;
                _netId := Tc2_System.F_CreateAmsNetId(nIds := _netIdArr);
                MasterNetId := _netId;
                NetIdMissing := FALSE;
                _step := 0;
            END_IF
        END_IF
    0:
        _fbStates(bExecute := FALSE);
        _fbStates(sNetId := _netId,
            pStateBuf := ADR(_stateBuf),
            cbBufLen := TO_UDINT(_slaveCount) * SIZEOF(Tc2_EtherCAT.ST_EcSlaveState),
            bExecute := (_slaveCount > 0));
        _step := 10;
    10:
        _fbStates(bExecute := FALSE);
        IF NOT _fbStates.bBusy THEN
            // Publish diagnostics every cycle so a failing read is visible.
            ReadOk := NOT _fbStates.bError;
            LastErrorId := _fbStates.nErrId;
            SlavesReported := _fbStates.nSlaves;
            IF NOT _fbStates.bError THEN
                FOR i := 1 TO _slaveCount DO
                    node := _firstSlaveNode + i - 1;
                    // pStateBuf is ARRAY[0..EC_MAX_SLAVES]: slave i lives at i-1.
                    // Decode the deviceState byte (AL state + flags) -> E_NodeState.
                    mapped := _M_MapSlaveState(DeviceState := _stateBuf[i - 1].deviceState);
                    // linkState low nibble = link condition; 0 = OK (EC_LINK_STATE_OK).
                    linkOk := (_stateBuf[i - 1].linkState AND 16#0F) = 0;
                    _pub^.M_SetNodeState(NodeIndex := node, State := mapped, LinkOk := linkOk);
                END_FOR
                // The master node's state is inferred from the read: it answered
                // ADS, so it is running. (A dedicated FB_EcGetMasterState read was
                // dropped to avoid a version-sensitive member name.)
                IF _masterNode >= 1 THEN
                    _pub^.M_SetNodeState(NodeIndex := _masterNode,
                        State := E_NodeState.OPERATIONAL, LinkOk := TRUE);
                END_IF
            ELSE
                // Master unreachable: mark the whole segment (and master) offline.
                _M_PublishAllOffline();
            END_IF
            _step := 20;
        END_IF
    20:
        _tPoll(IN := TRUE, PT := T#250MS);
        IF _tPoll.Q THEN
            _tPoll(IN := FALSE);
            _step := 0;
        END_IF
END_CASE
END_METHOD

// TRUE when the fieldbus is delivering a valid process image: the master read
// succeeded and every mapped slave is OPERATIONAL. This is the library-detected
// replacement for a project-declared "bus valid" flag — projects no longer wire
// their own RealBusOk. Derived from the last M_Refresh cycle (no extra I/O).
METHOD M_BusOk : BOOL
VAR
    i : INT;
END_VAR
M_BusOk := FALSE;
IF NOT _attached OR _fbStates.bError OR (_slaveCount < 1) THEN
    RETURN;
END_IF
FOR i := 1 TO _slaveCount DO
    // Zero-based buffer (see _stateBuf): slave i is at i-1. Fully operational iff
    // deviceState is exactly OP (no AL flag bits set).
    IF _stateBuf[i - 1].deviceState <> Tc2_EtherCAT.EC_DEVICE_STATE_OP THEN
        RETURN;  // any slave not OP -> bus not fully valid
    END_IF
END_FOR
M_BusOk := TRUE;
END_METHOD

// Fail-visible fallback: publish every mapped node (and the master) as OFFLINE.
// Used when the master cannot be reached and when its AmsNetId cannot be
// resolved -- an unknown bus must never look "operational" on the HMI.
METHOD PRIVATE _M_PublishAllOffline
VAR
    i : INT;
    node : INT;
END_VAR
IF NOT _attached THEN
    RETURN;
END_IF
FOR i := 1 TO _slaveCount DO
    node := _firstSlaveNode + i - 1;
    _pub^.M_SetNodeState(NodeIndex := node,
        State := E_NodeState.OFFLINE, LinkOk := FALSE);
END_FOR
IF _masterNode >= 1 THEN
    _pub^.M_SetNodeState(NodeIndex := _masterNode,
        State := E_NodeState.OFFLINE, LinkOk := FALSE);
END_IF
END_METHOD

// Decode an ST_EcSlaveState.deviceState byte (Beckhoff Tc2_EtherCAT, EtherCAT
// AL state machine) into the neutral E_NodeState the HMI renders.
//   low nibble  = AL state: INIT=1, PREOP=2, BOOTSTRAP=3, SAFEOP=4, OP=8
//   high nibble = flags:    ERROR=0x10, INVALID_VPRS=0x20, INITCMD_ERROR=0x40,
//                           DISABLED=0x80  -> any set is a fault.
// Source: infosys.beckhoff.com ST_EcSlaveState / EC_DEVICE_STATE_*.
METHOD PRIVATE _M_MapSlaveState : E_NodeState
VAR_INPUT
    DeviceState : BYTE;
END_VAR
// Any diagnostic flag bit (high nibble) overrides the AL state -> FAULT.
// After that check only the AL-state bits remain, so compare directly.
IF (DeviceState AND 16#F0) <> 0 THEN
    _M_MapSlaveState := E_NodeState.FAULT;
ELSIF DeviceState = Tc2_EtherCAT.EC_DEVICE_STATE_OP THEN
    _M_MapSlaveState := E_NodeState.OPERATIONAL;
ELSIF DeviceState = Tc2_EtherCAT.EC_DEVICE_STATE_SAFEOP THEN
    _M_MapSlaveState := E_NodeState.SAFEOP;
ELSIF DeviceState = Tc2_EtherCAT.EC_DEVICE_STATE_PREOP THEN
    _M_MapSlaveState := E_NodeState.PREOP;
ELSIF DeviceState = Tc2_EtherCAT.EC_DEVICE_STATE_INIT THEN
    _M_MapSlaveState := E_NodeState.INIT;
ELSE
    // BOOTSTRAP (0x03) or no state reported -> show as offline.
    _M_MapSlaveState := E_NodeState.OFFLINE;
END_IF
END_METHOD

END_FUNCTION_BLOCK

// ---- Connectivity/FB_IoTopologyPublisher.TcPOU
// Core §10.5.1 infrastructure service. Owns the reusable bounded-table,
// validation, health and diagnostic-join algorithms; project code supplies only
// physical topology metadata and live values. This is not a module tier.
FUNCTION_BLOCK FB_IoTopologyPublisher
VAR
    {attribute 'OPC.UA.DA' := '0'}
    _data : REFERENCE TO ST_FieldbusTopology;
    _attached : BOOL;
END_VAR

;

METHOD Setup : BOOL
VAR_INPUT
    DataRef : REFERENCE TO ST_FieldbusTopology;
    ResetData : BOOL;
END_VAR
VAR
    n, c : INT;
END_VAR
_data REF= DataRef;
_attached := __ISVALIDREF(_data);
IF _attached AND ResetData THEN
    _data.NodeCount := 0;
    _data.MappingValid := TRUE;
    _data.MappingDiagnostic := '';
    FOR n := 1 TO PL_Fraktal.MAX_BUS_NODES DO
        _data.Nodes[n].Name := '';
        _data.Nodes[n].DescriptionKey := '';
        _data.Nodes[n].TypeId := '';
        _data.Nodes[n].Address := '';
        _data.Nodes[n].ParentIdx := 0;
        _data.Nodes[n].ChannelCount := 0;
        FOR c := 1 TO PL_Fraktal.MAX_NODE_CHANNELS DO
            _data.Nodes[n].Channels[c].Name := '';
            _data.Nodes[n].Channels[c].Path := '';
        END_FOR
    END_FOR
ELSIF _attached THEN
    ;
ELSE
    _attached := FALSE;
END_IF
Setup := _attached;
END_METHOD

METHOD M_DefineNode : BOOL
VAR_INPUT
    Index : INT;
    Name : STRING(80);
    DescriptionKey : STRING(160);
    TypeId : STRING(80);
    Address : STRING(40);
    ParentIndex : INT;
END_VAR
M_DefineNode := FALSE;
IF NOT _attached THEN
    RETURN;
ELSE
    ;
END_IF
IF (Index < 1) OR (Index > PL_Fraktal.MAX_BUS_NODES)
OR (Name = '') OR (Address = '')
OR (ParentIndex < 0) OR (ParentIndex >= Index) THEN
    _M_Reject(Text := 'std.error.fieldbusNodeMappingInvalid');
    RETURN;
ELSE
    ;
END_IF
_data.Nodes[Index].Name := Name;
_data.Nodes[Index].DescriptionKey := DescriptionKey;
_data.Nodes[Index].TypeId := TypeId;
_data.Nodes[Index].Address := Address;
_data.Nodes[Index].ParentIdx := ParentIndex;
IF Index > _data.NodeCount THEN
    _data.NodeCount := Index;
ELSE
    ;
END_IF
M_DefineNode := TRUE;
END_METHOD

METHOD M_DefineDigitalChannel : BOOL
VAR_INPUT
    NodeIndex : INT;
    ChannelIndex : INT;
    Tag : STRING(80);
    DescriptionKey : STRING(160);
    Address : STRING(80);
    Path : STRING(255);
    ModulePath : STRING(255);
    Dir : E_ChannelDir;
END_VAR
M_DefineDigitalChannel := FALSE;
IF NOT _attached THEN
    RETURN;
ELSE
    ;
END_IF
IF (NodeIndex < 1) OR (NodeIndex > _data.NodeCount)
OR (ChannelIndex < 1) OR (ChannelIndex > PL_Fraktal.MAX_NODE_CHANNELS)
OR (Tag = '') OR (DescriptionKey = '') OR (Address = '')
OR (Path = '') OR (ModulePath = '') THEN
    _M_Reject(Text := 'std.error.fieldbusChannelMappingInvalid');
    RETURN;
ELSE
    ;
END_IF
_data.Nodes[NodeIndex].Channels[ChannelIndex].Name := Tag;
_data.Nodes[NodeIndex].Channels[ChannelIndex].DescriptionKey := DescriptionKey;
_data.Nodes[NodeIndex].Channels[ChannelIndex].Address := Address;
_data.Nodes[NodeIndex].Channels[ChannelIndex].Path := Path;
_data.Nodes[NodeIndex].Channels[ChannelIndex].ModulePath := ModulePath;
_data.Nodes[NodeIndex].Channels[ChannelIndex].Dir := Dir;
_data.Nodes[NodeIndex].Channels[ChannelIndex].Kind := E_ChannelKind.DIGITAL;
_data.Nodes[NodeIndex].Channels[ChannelIndex].Quality := TRUE;
IF ChannelIndex > _data.Nodes[NodeIndex].ChannelCount THEN
    _data.Nodes[NodeIndex].ChannelCount := ChannelIndex;
ELSE
    ;
END_IF
M_DefineDigitalChannel := TRUE;
END_METHOD

METHOD M_SetDigitalValue : BOOL
VAR_INPUT
    NodeIndex : INT;
    ChannelIndex : INT;
    Value : BOOL;
END_VAR
M_SetDigitalValue := FALSE;
IF _attached AND (NodeIndex >= 1) AND (NodeIndex <= _data.NodeCount)
AND (ChannelIndex >= 1) AND (ChannelIndex <= _data.Nodes[NodeIndex].ChannelCount) THEN
    _data.Nodes[NodeIndex].Channels[ChannelIndex].BoolValue := Value;
    M_SetDigitalValue := TRUE;
ELSE
    _M_Reject(Text := 'std.error.fieldbusValueMappingInvalid');
END_IF
END_METHOD

// Legacy/fallback: force one health verdict on every node. Kept for transports
// or projects that cannot read per-node bus state (e.g. no fieldbus master).
// Prefer M_SetNodeState so the HMI shows each node's REAL state.
METHOD M_SetAllHealth
VAR_INPUT
    Healthy : BOOL;
END_VAR
VAR
    n, c : INT;
END_VAR
IF _attached THEN
    FOR n := 1 TO _data.NodeCount DO
        _data.Nodes[n].LinkOk := Healthy;
        IF Healthy THEN
            _data.Nodes[n].State := E_NodeState.OPERATIONAL;
        ELSE
            _data.Nodes[n].State := E_NodeState.FAULT;
        END_IF
        FOR c := 1 TO _data.Nodes[n].ChannelCount DO
            _data.Nodes[n].Channels[c].Quality := Healthy;
        END_FOR
    END_FOR
ELSE
    ;
END_IF
END_METHOD

// Core §10.5.1: publish ONE node's real fieldbus state, independent of any
// control/safety verdict. State is the neutral E_NodeState the HMI renders
// (INIT/PREOP/SAFEOP/OPERATIONAL/FAULT/OFFLINE); LinkOk mirrors the physical
// link. Channel Quality follows link health (a down node's values are stale).
// The caller derives State/LinkOk from the actual bus master (see FB_EcBusHealth
// for EtherCAT); node state is NOT conditioned by Control-On or safety.
METHOD M_SetNodeState : BOOL
VAR_INPUT
    NodeIndex : INT;
    State : E_NodeState;
    LinkOk : BOOL;
END_VAR
VAR
    c : INT;
END_VAR
M_SetNodeState := FALSE;
IF _attached AND (NodeIndex >= 1) AND (NodeIndex <= _data.NodeCount) THEN
    _data.Nodes[NodeIndex].State := State;
    _data.Nodes[NodeIndex].LinkOk := LinkOk;
    FOR c := 1 TO _data.Nodes[NodeIndex].ChannelCount DO
        _data.Nodes[NodeIndex].Channels[c].Quality := LinkOk;
    END_FOR
    M_SetNodeState := TRUE;
ELSE
    ;
END_IF
END_METHOD

METHOD M_BeginDiagnosticRefresh
VAR
    n, c : INT;
END_VAR
IF _attached THEN
    FOR n := 1 TO _data.NodeCount DO
        FOR c := 1 TO _data.Nodes[n].ChannelCount DO
            _data.Nodes[n].Channels[c].FaultActive := FALSE;
            _data.Nodes[n].Channels[c].Diagnostic := '';
        END_FOR
    END_FOR
ELSE
    ;
END_IF
END_METHOD

METHOD M_ApplyDiagnostic
VAR_INPUT
    Diagnostic : ST_Diagnostic;
END_VAR
IF Diagnostic.IoTag <> '' THEN
    M_ApplyDiagnosticToTag(Diagnostic := Diagnostic, Tag := Diagnostic.IoTag);
ELSE
    ;
END_IF
END_METHOD

METHOD M_ApplyDiagnosticToTag
VAR_INPUT
    Diagnostic : ST_Diagnostic;
    Tag : STRING(80);
END_VAR
VAR
    n, c : INT;
END_VAR
IF _attached AND (Tag <> '') THEN
    FOR n := 1 TO _data.NodeCount DO
        FOR c := 1 TO _data.Nodes[n].ChannelCount DO
            IF _data.Nodes[n].Channels[c].Name = Tag THEN
                _data.Nodes[n].Channels[c].FaultActive := TRUE;
                _data.Nodes[n].Channels[c].Diagnostic := Diagnostic.Description;
            ELSE
                ;
            END_IF
        END_FOR
    END_FOR
ELSE
    ;
END_IF
END_METHOD

METHOD M_Validate : BOOL
VAR
    n, c, n2, c2 : INT;
END_VAR
M_Validate := FALSE;
IF NOT _attached OR (_data.NodeCount < 1) THEN
    _M_Reject(Text := 'std.error.fieldbusTopologyEmpty');
    RETURN;
ELSE
    ;
END_IF
IF NOT _data.MappingValid THEN
    RETURN; // preserve the first registration/value mapping failure
ELSE
    ;
END_IF
FOR n := 1 TO _data.NodeCount DO
    IF (_data.Nodes[n].Name = '') OR (_data.Nodes[n].Address = '') THEN
        _M_Reject(Text := 'std.error.fieldbusNodeMappingInvalid');
        RETURN;
    ELSE
        ;
    END_IF
    FOR c := 1 TO _data.Nodes[n].ChannelCount DO
        IF (_data.Nodes[n].Channels[c].Name = '')
        OR (_data.Nodes[n].Channels[c].Address = '')
        OR (_data.Nodes[n].Channels[c].Path = '')
        OR (_data.Nodes[n].Channels[c].ModulePath = '') THEN
            _M_Reject(Text := 'std.error.fieldbusChannelMappingInvalid');
            RETURN;
        ELSE
            ;
        END_IF
        FOR n2 := n TO _data.NodeCount DO
            FOR c2 := 1 TO _data.Nodes[n2].ChannelCount DO
                IF ((n2 > n) OR (c2 > c))
                AND ((_data.Nodes[n].Channels[c].Name = _data.Nodes[n2].Channels[c2].Name)
                  OR (_data.Nodes[n].Channels[c].Path = _data.Nodes[n2].Channels[c2].Path)) THEN
                    _M_Reject(Text := 'std.error.fieldbusChannelIdentityDuplicate');
                    RETURN;
                ELSE
                    ;
                END_IF
            END_FOR
        END_FOR
    END_FOR
END_FOR
_data.MappingValid := TRUE;
_data.MappingDiagnostic := '';
M_Validate := TRUE;
END_METHOD

METHOD PRIVATE _M_Reject
VAR_INPUT
    Text : STRING(255);
END_VAR
IF _attached THEN
    _data.MappingValid := FALSE;
    _data.MappingDiagnostic := Text;
ELSE
    ;
END_IF
END_METHOD

END_FUNCTION_BLOCK

// ---- Connectivity/FB_LocalStationConfig.TcPOU
// Core §3.8a — DEFAULT station-config provider: in-PLC PERSISTENT records, editable
// locally over OPC UA (§3.10). Remote sources (asset system, MES) substitute later
// through I_StationConfig without touching module code (O1, O6).
FUNCTION_BLOCK FB_LocalStationConfig IMPLEMENTS I_StationConfig
VAR PERSISTENT
    _n : INT;
END_VAR
VAR
    _keys : ARRAY[1..PL_Fraktal.MAX_STATIONCFG] OF STRING(80);
    _ptr  : ARRAY[1..PL_Fraktal.MAX_STATIONCFG] OF PVOID;
    _size : ARRAY[1..PL_Fraktal.MAX_STATIONCFG] OF UDINT;
END_VAR

// no cyclic body

METHOD Load : BOOL
VAR_INPUT
    Key : STRING;
    pCfg : PVOID;
    Size : UDINT;
END_VAR
VAR
    i : INT;
END_VAR
Load := FALSE;
FOR i := 1 TO _n DO
    IF (_keys[i] = Key) AND (_size[i] = Size) AND (pCfg <> 0) THEN
        MEMCPY(destAddr := pCfg, srcAddr := _ptr[i], n := Size);
        Load := TRUE;
        RETURN;
    END_IF
END_FOR
END_METHOD

METHOD Store : BOOL
VAR_INPUT
    Key : STRING;
    pCfg : PVOID;
    Size : UDINT;
END_VAR
VAR
    i : INT;
END_VAR
Store := FALSE;
FOR i := 1 TO _n DO
    IF (_keys[i] = Key) AND (_size[i] = Size) AND (pCfg <> 0) THEN
        MEMCPY(destAddr := _ptr[i], srcAddr := pCfg, n := Size);   // persists (registered targets live in persistent areas)
        Store := TRUE;
        RETURN;
    END_IF
END_FOR
END_METHOD

// application wiring: bind a module's PERSISTENT StationCfg to a key
METHOD Register : BOOL
VAR_INPUT
    Key : STRING(80);
    pData : PVOID;
    Size : UDINT;
END_VAR
IF (_n >= PL_Fraktal.MAX_STATIONCFG) OR (pData = 0) THEN
    Register := FALSE;
    RETURN;
END_IF
_n := _n + 1;
_keys[_n] := Key;
_ptr[_n] := pData;
_size[_n] := Size;
Register := TRUE;
END_METHOD

END_FUNCTION_BLOCK

// ---- DeviceCMs/FB_TcpCodeReaderCM.TcPOU
// Core §3.15.1a — CATEGORY CM: triggered TCP/ASCII code reader (barcode/DMC),
// vendor-neutral. Configure for most readers; extend only for special features.
// Optional match-code verification: ParCmd.MatchCode <> ''.
// Publishes: ParCfg, ParCmd, OutCmd, OutImm. Feeds Annex E.
FUNCTION_BLOCK FB_TcpCodeReaderCM EXTENDS FB_AsciiDeviceCM
VAR_INPUT
    ParCfg : ST_TcpCodeReaderParCfg;
    ParCmd : ST_TcpCodeReaderParCmd;
END_VAR
VAR_OUTPUT
    OutCmd : ST_TcpCodeReaderOutCmd;
    OutImm : ST_TcpCodeReaderOutImm;
END_VAR
VAR
    _done : BOOL;
    _sent : BOOL;
END_VAR

Cyclic();

METHOD Setup : BOOL
VAR_INPUT
    Name : STRING(80);
    Chan : I_ByteChannel;
    DevHost : STRING(80);
    DevPort : UINT;
END_VAR
_M_SetName(Name);
_M_PublishCommand(Value := 1, Label := 'std.command.triggerRead');
ParCfg.Host := DevHost;
ParCfg.Port := DevPort;
Setup := SetupDevice(Chan := Chan, DevHost := DevHost, DevPort := DevPort);
END_METHOD

METHOD PROTECTED _M_Dispatch
IF _manualReq THEN
    _manualReq := FALSE;
    IF _manualCmd = 1 THEN
        _sent := SendRequest(Text := ParCfg.TriggerCmd);
        IF _sent THEN OutCmd.Code := ''; OutCmd.NoRead := FALSE; OutCmd.MatchOk := FALSE; END_IF
    ELSE
        _M_Fault(E_Reason.UNSUPPORTED_COMMAND, 'std.error.unsupportedCodeReaderCommand');
        RETURN;
    END_IF
END_IF
IF Execute THEN
    IF NOT _sent THEN
        _M_TagCommand(Id := 1, Label := 'std.command.triggerRead');
        _sent := SendRequest(Text := ParCfg.TriggerCmd);
        IF _sent THEN
            OutCmd.Code := '';
            OutCmd.NoRead := FALSE;
            OutCmd.MatchOk := FALSE;
        END_IF
    ELSIF _done THEN
        _sent := FALSE;
        _done := FALSE;
        _M_Complete();
    END_IF
ELSE
    _sent := FALSE;
    _done := FALSE;
END_IF
END_METHOD

METHOD PROTECTED OnCyclic : DINT
OnCyclic := SUPER^.OnCyclic();
Host := ParCfg.Host;
Port := ParCfg.Port;
Terminator := ParCfg.Terminator;
RespTimeout := ParCfg.RespTimeout;
OutImm.LinkState := LinkState;
OutImm.LastResponse := LastResponse;
OutImm.Diagnostic := Status.Diagnostic;
END_METHOD

// generic read parse: NoReadText or the decoded symbol; optional match verify.
METHOD PROTECTED _M_OnResponse
VAR_INPUT
    Response : STRING(255);
END_VAR
OutCmd.NoRead := (Response = ParCfg.NoReadText);
IF OutCmd.NoRead THEN OutCmd.Code := ''; END_IF
IF NOT OutCmd.NoRead THEN
    OutCmd.Code := Response;             // -> traceability (Annex E)
END_IF
IF ParCmd.MatchCode <> '' THEN
    OutCmd.MatchOk := (NOT OutCmd.NoRead) AND (Response = ParCmd.MatchCode);
ELSE
    OutCmd.MatchOk := NOT OutCmd.NoRead;
END_IF
_done := TRUE;
END_METHOD

METHOD PROTECTED _M_PublishStatus
SUPER^._M_PublishStatus();
OutImm.Diagnostic := Status.Diagnostic;
END_METHOD

END_FUNCTION_BLOCK
